{attribute 'qualified_only'}
{attribute 'strict'}
{attribute 'to_string'}
TYPE E_MainStateMachine :
(
	Init := 0,
    step0,
    step1,
    step2,
    step3,
    step4,
    TipStep,
    error
);
END_TYPE

(* stored: Version 1.1.0.1
   DUT E_MainStateMachine: Id {bc461f51-9910-0c15-21e8-451f8e4edb44} *)
